FUNCTION_BLOCK ABSTRACT ComponentBase IMPLEMENTS IPluginRunner, IPlugin
VAR
	i_ComponentBase : ComponentBaseInternal;
END_VAR

Run();

METHOD Cyclic
//This method is meant to be overridden to contain any cyclic function block calls
END_METHOD

METHOD Init : BOOL
VAR_INPUT
END_VAR
VAR
	nData : UDINT;
	pData : PVOID;
END_VAR
InitComplete();
END_METHOD

METHOD InitComplete
VAR_INPUT
END_VAR
i_ComponentBase._initDone := TRUE;
LogMessage( 0, 'Init Complete');
END_METHOD

METHOD RegisterPlugin
VAR_INPUT
	plugin : IPlugin;
END_VAR
i_ComponentBase._plugins.RegisterPlugin(plugin);
END_METHOD

METHOD Run : BOOL
VAR_INPUT
END_VAR
//If we aren't initialized, call init
IF NOT i_ComponentBase._initDone THEN
	
	//Init any derived classes
	THIS^.Init();
	
END_IF

runPlugins();

//Init() was successful, call cyclic
IF i_ComponentBase._initDone THEN
	
	THIS^.Running();

END_IF
END_METHOD

METHOD Running : BOOL
VAR_INPUT
END_VAR
//Run the main code
THIS^.Simulation();

THIS^.Cyclic();
END_METHOD

METHOD PRIVATE runPlugins
i_ComponentBase._plugins.runPlugins();
END_METHOD

METHOD Simulation : BOOL
VAR_INPUT
END_VAR
END_METHOD

END_FUNCTION_BLOCK

(* stored: Version 1.1.0.1, ProductVersion 3.1.4024.12
   POU ComponentBase: Id {fd84c14d-786e-4719-a893-d07044f55331}, SpecialFunc None
   Folder API: Id {c262686b-39a8-47b3-a436-2f37f829fd3b}
   Folder ApplicationOverrides: Id {f2009942-3f7f-4941-bfa7-741ffc14e21c}
   Folder Internal: Id {e1a9125c-f3ee-490f-ba83-a56d67f46885}
   Method Cyclic: Id {f52824b0-33e3-4c0b-be35-3a5b4aa4be2f}
   Method Init: Id {e101f04f-5e1f-4e3c-b777-2115fc0732ac}
   Method InitComplete: Id {87aa42d7-dc57-4645-9c0e-f16722b7922f}
   Method RegisterPlugin: Id {571843c1-23e2-4fb3-8310-25661dcfe26f}
   Method Run: Id {261da83f-aad6-40a0-bf8a-54e818a518b0}
   Method Running: Id {2a550c20-dd34-4807-bd60-3c34c3be85bf}
   Method runPlugins: Id {98b78174-293e-4815-ac54-043bcc5693a6}
   Method Simulation: Id {86233419-db64-4072-8f39-139f044b5b04} *)
